// TIA Portal V20 export
// export: Created 2026-04-11T06:02:29.9965815Z, ExportSetting WithDefaults, DisplayName Totally Integrated Automation Portal, DisplayVersion V20, DisplayName TIA Portal Openness, DisplayVersion V20, DisplayName TIA Portal Version Control Interface, DisplayVersion V20, DisplayName STEP 7 Professional, DisplayVersion V20, DisplayName STEP 7 Safety, DisplayVersion V20, DisplayName WinCC Basic/Comfort/Advanced, DisplayVersion V20, DisplayName WinCC Unified, DisplayVersion V20
TYPE "udtError_Valve"
// stored: IsFailsafeCompliant false
   STRUCT
      NoHomeFeedback { ExternalWritable := 'False'} : Bool;   // Home position feedback not active
      NoWorkFeedback { ExternalWritable := 'False'} : Bool;   // Work position feedback not active
      HomeFeedbackStillActive { ExternalWritable := 'False'} : Bool;   // Home position feedback still active
      WorkFeedbackStillActive { ExternalWritable := 'False'} : Bool;   // Work position feedback still active
   END_STRUCT;
END_TYPE
